RoboDK station: mirobot.rdk

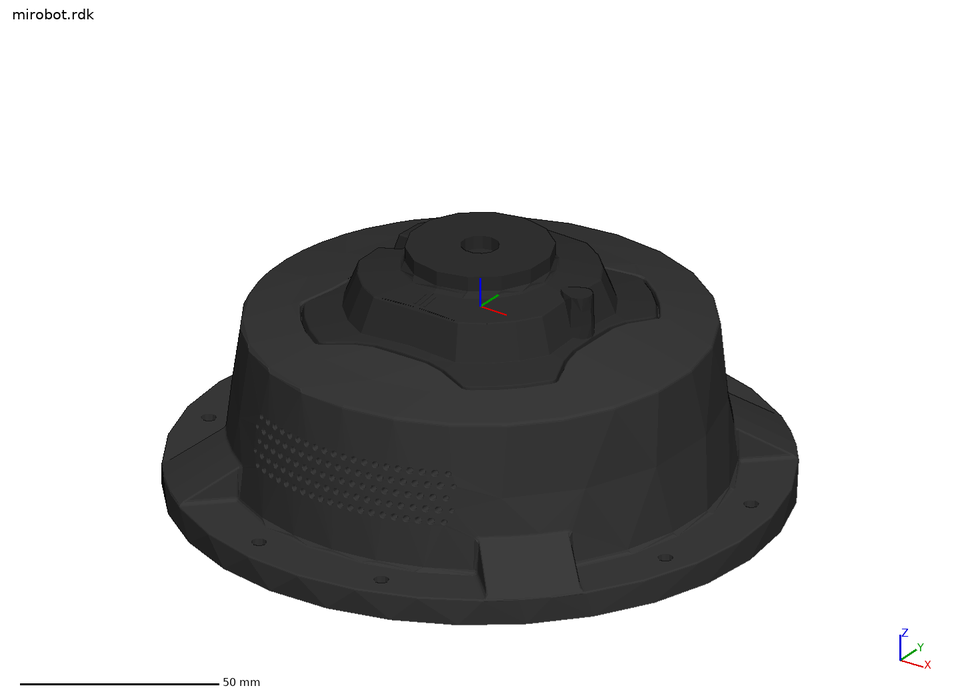
[picture v0: the station drawn from its stored meshes, robots at their saved joint values, targets as dots, program paths as lines]
Station mirobot (saved by RoboDK 5.6.3). Poses are relative to the parent item; angles as X-Y-Z fixed-axis rotations.
  - frame Wlkata Mirobot Base at (0, 0, 0) mm
    - robot Wlkata Mirobot: 6 axes, payload 0.4 kg, reach 315 mm, repeatability 0.2 mm, weight 1.5 kg
        joint limits [-100, -60, -180, -180, -180, -180] to [100, 90, 50, 180, 50, 180]; home [0, 0, 0, 0, 0, 0]; saved at [3, 22.2, -15.05, 0, -7.18, 10.74]
      - tool intel_realsense, TCP at (0, 0, 0) mm, rotated rx 180 ry 0 rz 180 deg
      - tool tool, TCP at (0, 0, 0) mm, rotated rx 180 ry 0 rz 180 deg
  - frame Ground at (238.1, -17.49, -50) mm
  - frame Crack at (256.54, 41.87, 44.46) mm
